{attribute 'qualified_only'}
VAR_GLOBAL
	bChamber1_Endpoint1_DoorClosed : BOOL;
	bChamber1_VacuumOn : BOOL;
	
	bRobotIsInChamber1 : BOOL;
END_VAR

(* stored: Version 1.1.0.1, ProductVersion 3.1.4026.18
   GVL GVL_ShareMemory: Id {0ac7dcd6-2d9a-4945-95c6-b1033d0f2923} *)
